(* PLC project Programme MGS_2-07_refactorJOY.project, CODESYS CODESYS V3.5 SP19 Patch 1 *)
(* stored: creationDateTime 2026-06-29T23:37:40.9386598, modificationDateTime 2026-06-29T22:49:33.424 *)

FUNCTION_BLOCK FB_AxisScale
  VAR_INPUT
    RawIn : INT;  (* Valeur brute (0..10000) *)
    Neutral : INT;  (* Point milieu calibré *)
    Deadband : REAL;  (* Zone morte en % *)
  END_VAR
  VAR_OUTPUT
    OutPct : REAL;  (* Valeur finale (-100.0..100.0) *)
  END_VAR
  VAR
    Delta : REAL;
  END_VAR

            IF RawIn >= Neutral THEN
    Delta := INT_TO_REAL(10000 - Neutral);
    IF Delta > 0.0 THEN
        OutPct := (INT_TO_REAL(RawIn - Neutral) / Delta) * 100.0;
    ELSE
        OutPct := 0.0;
    END_IF;
ELSE
    Delta := INT_TO_REAL(Neutral);
    IF Delta > 0.0 THEN
        OutPct := (INT_TO_REAL(RawIn - Neutral) / Delta) * 100.0;
    ELSE
        OutPct := 0.0;
    END_IF;
END_IF;

IF ABS(OutPct) <= Deadband THEN
    OutPct := 0.0;
END_IF;
          
END_FUNCTION_BLOCK
